ABB RobotStudio station: VInRoS_ROB_1_Project.rspag

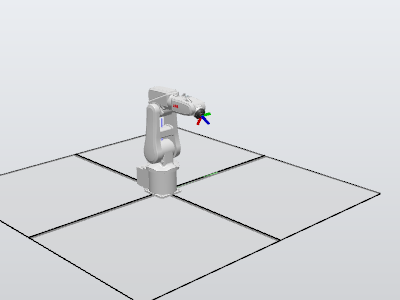
--- station ---
Station VInRoS_ROB_1_Project (saved by RobotStudio 23.2.10478.1)
Controller Controller1
  mechanical unit ROB_1: IRB120_3_58__01, 6 joints, base frame (0, 0, 0) mm
Layout (positions relative to the parent item):
  - IRB120_3_58__01 [mechanism, from %ABB.RobotStudio.Models.IRB120%\IRB120_3_58_G_01.rslib] at (0, 0, 0) mm; joint values [0, 0, 0, 0, 0.5236, 0] (rad or m)

--- Controller Data/Controller1/RAPID/TASK1/PROGMOD/Module1.mod ---
MODULE Module1
    ! ## =========================================================================== ##
    ! MIT License
    ! Copyright (c) 2021 Roman Parak
    ! Permission is hereby granted, free of charge, to any person obtaining a copy
    ! of this software and associated documentation files (the "Software"), to deal
    ! in the Software without restriction, including without limitation the rights
    ! to use, copy, modify, merge, publish, distribute, sublicense, and/or sell
    ! copies of the Software, and to permit persons to whom the Software is
    ! furnished to do so, subject to the following conditions:
    ! The above copyright notice and this permission notice shall be included in all
    ! copies or substantial portions of the Software.
    ! THE SOFTWARE IS PROVIDED "AS IS", WITHOUT WARRANTY OF ANY KIND, EXPRESS OR
    ! IMPLIED, INCLUDING BUT NOT LIMITED TO THE WARRANTIES OF MERCHANTABILITY,
    ! FITNESS FOR A PARTICULAR PURPOSE AND NONINFRINGEMENT. IN NO EVENT SHALL THE
    ! AUTHORS OR COPYRIGHT HOLDERS BE LIABLE FOR ANY CLAIM, DAMAGES OR OTHER
    ! LIABILITY, WHETHER IN AN ACTION OF CONTRACT, TORT OR OTHERWISE, ARISING FROM,
    ! OUT OF OR IN CONNECTION WITH THE SOFTWARE OR THE USE OR OTHER DEALINGS IN THE
    ! SOFTWARE.
    ! ## =========================================================================== ##
    ! Author   : Roman Parak
    ! Email    : Roman.Parak@outlook.com
    ! Github   : https://github.com/rparak
    ! File Name: T_ROB_MAIN_CTRL/Module1.mod
    ! ## =========================================================================== ##

    ! Description: !
    !   The main command structure for robot control !
    RECORD robot_command_main_str
        num start;
        num stop;
        num id;
        num update;
    ENDRECORD

    ! Description: !
    !   The main structure of the robot control parameters !
    RECORD robot_param_main_str
        num Trajectory_Size;
    ENDRECORD

    ! Description: !
    !   The main structure of robot status information !
    RECORD robot_status_str
        num in_position; ! Signaling when the robot is in the target position
        num active;      ! Signaling when everything on the robot's side is fine
        num id;          ! Identification number of the current state of the robot
        num update_done; ! Signaling when the parameter update is completed successfully
        num actual_trajectory_id;
    ENDRECORD

    ! Description: !
    !   The main structure of PLC status information !
    RECORD plc_status_str
        num active; ! Signaling when everything on the PC's (PLC) side is OK
        num update_done;
    ENDRECORD

    ! Description: !
    !   The main structure of status information !
    RECORD status_main_str
        plc_status_str plc;
        robot_status_str robot;
    ENDRECORD

    ! Description: !
    !   The main structure of internal values !
    RECORD internal_main_str
        num actual_state;               ! Current state in the main state machine
        num previous_state;             ! Previous state in the main state machine
        num accuracy_factor;            ! Accuracy factor for value conversion (Default)
        num accuracy_factor_QUATERNION; ! Accuracy factor for value conversion (QUATERNION)
        num actual_trajectory_id;
    ENDRECORD

    ! Description: !
    !   The main control structure of the robot !
    RECORD robot_ctrl_str
        robot_param_main_str parameter; ! Robot control parameters
        robot_command_main_str command; ! Command structure for robot control
        status_main_str status;         ! Robot status information
        internal_main_str internal;     ! Internal values
    ENDRECORD

    ! Call Main Structure
    PERS robot_ctrl_str rm_str;

    ! Joint Position Data
    PERS jointtarget J_Position{100};

    ! TCP Position Data
    PERS robtarget TCP_Position{100};

    ! Joint Speed Data
    PERS speeddata Speed{100};

    ! Joint Zone Data
    PERS zonedata Zone{100};

    ! Characteristics of a robotic tool (end-effector / gripper)
    PERS tooldata robTool;

    VAR num aux_trajectory_index_var;

    ! Description:               !
    !   Program Main Cycle:      !
    !       Type        : Normal !
    !       TrustLeve   : N/A    !
    !       Motion Task : YES    !
    PROC Main()
        TEST ROB_ST_MAIN_ID_PROFINET_OUT
            CASE 10: ! INITIALIZATION STATE !
                ! Description: !
                !   Initialization state to check everything on the PC's (PLC) side and activation to control !

                ! Initialize the internal value of the accuracy conversion factor
                rm_str.internal.accuracy_factor            := 100;
                rm_str.internal.accuracy_factor_QUATERNION := 100000000;

                SetDO ROB_ST_ACTIVE_PROFINET_OUT, 1;

                IF PLC_ST_ACTIVE_PROFINET_IN = 1 THEN
                    ! Wait State {rm_str.status.plc.ModuleOK = TRUE -> Everything on the PC's (PLC) side is OK}
                    SetGO ROB_ST_MAIN_ID_PROFINET_OUT, 20;
                ENDIF

            CASE 20: ! WAIT STATE !
                ! Description: !
                !   State of waiting for command with index from the PC's (PLC) !

                aux_trajectory_index_var := 0;

                IF PLC_CMD_START_PROFINET_IN = 1 AND PLC_CMD_MAIN_ID_PROFINET_IN = 1 THEN
                    SetDO ROB_ST_IN_POS_PROFINET_OUT, 0;
                    ! Move Joint (Absolute)
                    SetGO ROB_ST_MAIN_ID_PROFINET_OUT, 30;
                ELSEIF PLC_CMD_START_PROFINET_IN = 1 AND PLC_CMD_MAIN_ID_PROFINET_IN = 2 THEN
                    SetDO ROB_ST_IN_POS_PROFINET_OUT, 0;
                    ! Move Linear
                    SetGO ROB_ST_MAIN_ID_PROFINET_OUT, 40;
                ENDIF

                IF PLC_ST_ACTIVE_PROFINET_IN = 0 THEN
                    ! Initialization State {rm_str.PLC_ModuleOK = FALSE -> There is some problem with the PC's (PLC)}
                    SetGO ROB_ST_MAIN_ID_PROFINET_OUT, 10;
                ENDIF

            CASE 30: ! MOVE JOINT ABSOLUTE STATE - EXECUTE !
                ! Description: !
                !   Control Function (MoveAbsJ): Moves the robot to an absolute joint position !

                IF aux_trajectory_index_var = PLC_TRAJ_SIZE_PROFINET_IN THEN
                    SetDO ROB_ST_IN_POS_PROFINET_OUT, 1;
                    SetGO ROB_ST_MAIN_ID_PROFINET_OUT, 20;
                ELSE
                    SetGO ROB_MOTION_TRAJ_ID_PROFINET_OUT, aux_trajectory_index_var;
                    MoveAbsJ J_Position{aux_trajectory_index_var + 1}\NoEOffs, Speed{aux_trajectory_index_var + 1}, Zone{aux_trajectory_index_var + 1}, robTool\WObj:=wobj0;
                    aux_trajectory_index_var := aux_trajectory_index_var + 1;
                ENDIF

            CASE 40: ! MOVE CARTESIAN STATE - EXECUTE !
                ! Description: !
                !   Control Function (MoveL): Moves the tool center point (TCP) linearly !

                IF aux_trajectory_index_var = PLC_TRAJ_SIZE_PROFINET_IN THEN
                    SetDO ROB_ST_IN_POS_PROFINET_OUT, 1;
                    SetGO ROB_ST_MAIN_ID_PROFINET_OUT, 20;
                ELSE
                    SetGO ROB_MOTION_TRAJ_ID_PROFINET_OUT, aux_trajectory_index_var;
                    MoveL TCP_Position{aux_trajectory_index_var + 1}, Speed{aux_trajectory_index_var + 1}, Zone{aux_trajectory_index_var + 1}, robTool\WObj:=wobj0;
                    aux_trajectory_index_var := aux_trajectory_index_var + 1;
                ENDIF
        ENDTEST
    ENDPROC

    PROC ER_Reset_Parameters_MAIN_CTRL()
        ! Description:                                                   !
        !   Event routine function (non-parametric) for parameter reset. !
        !       Note: Configuration / Controller / Event Routine         !

        SetGO ROB_ST_MAIN_ID_PROFINET_OUT, 10;
        SetGO ROB_ST_UPT_ID_PROFINET_OUT, 10;

        ! Main Control Structure
        rm_str := [[0],[0,0,0,0],[[0,0],[0,0,0,0,0]],[0,0,0,0,0]];

        ! Characteristics of a robotic tool (end-effector / gripper)
        robTool := [TRUE,[[0,0,0],[1,0,0,0]],[0.001,[0,0,0.001],[1,0,0,0],0,0,0]];
	ENDPROC

    PROC ER_Reset_Parameters_Stopped()
        ! Description:                                                   !
        !   Event routine function (non-parametric) to reset parameters  !
        !   when the program is stopped.                                 !
        !       Note: Configuration / Controller / Event Routine         !

        SetDO ROB_ST_IN_POS_PROFINET_OUT, 1;
        SetGO ROB_ST_MAIN_ID_PROFINET_OUT, 10;
    ENDPROC
ENDMODULE

--- Controller Data/Controller1/RAPID/TASK2/PROGMOD/Module1.mod ---
MODULE Module1
    ! ## =========================================================================== ##
    ! MIT License
    ! Copyright (c) 2021 Roman Parak
    ! Permission is hereby granted, free of charge, to any person obtaining a copy
    ! of this software and associated documentation files (the "Software"), to deal
    ! in the Software without restriction, including without limitation the rights
    ! to use, copy, modify, merge, publish, distribute, sublicense, and/or sell
    ! copies of the Software, and to permit persons to whom the Software is
    ! furnished to do so, subject to the following conditions:
    ! The above copyright notice and this permission notice shall be included in all
    ! copies or substantial portions of the Software.
    ! THE SOFTWARE IS PROVIDED "AS IS", WITHOUT WARRANTY OF ANY KIND, EXPRESS OR
    ! IMPLIED, INCLUDING BUT NOT LIMITED TO THE WARRANTIES OF MERCHANTABILITY,
    ! FITNESS FOR A PARTICULAR PURPOSE AND NONINFRINGEMENT. IN NO EVENT SHALL THE
    ! AUTHORS OR COPYRIGHT HOLDERS BE LIABLE FOR ANY CLAIM, DAMAGES OR OTHER
    ! LIABILITY, WHETHER IN AN ACTION OF CONTRACT, TORT OR OTHERWISE, ARISING FROM,
    ! OUT OF OR IN CONNECTION WITH THE SOFTWARE OR THE USE OR OTHER DEALINGS IN THE
    ! SOFTWARE.
    ! ## =========================================================================== ##
    ! Author   : Roman Parak
    ! Email    : Roman.Parak@outlook.com
    ! Github   : https://github.com/rparak
    ! File Name: T_PLC_ROB_PROFINET/Module1.mod
    ! ## =========================================================================== ##


    ! Description: !
    !   The main command structure for robot control !
    RECORD robot_command_main_str
        num start;
        num stop;
        num id;
        num update;
    ENDRECORD

    ! Description: !
    !   The main structure of the robot control parameters !
    RECORD robot_param_main_str
        num Trajectory_Size;
    ENDRECORD

    ! Description: !
    !   The main structure of robot status information !
    RECORD robot_status_str
        num in_position; ! Signaling when the robot is in the target position
        num active;      ! Signaling when everything on the robot's side is fine
        num id;          ! Identification number of the current state of the robot
        num update_done; ! Signaling when the parameter update is completed successfully
        num actual_trajectory_id;
    ENDRECORD

    ! Description: !
    !   The main structure of PLC status information !
    RECORD plc_status_str
        num active; ! Signaling when everything on the PC's (PLC) side is OK
        num update_done;
    ENDRECORD

    ! Description: !
    !   The main structure of status information !
    RECORD status_main_str
        plc_status_str plc;
        robot_status_str robot;
    ENDRECORD

    ! Description: !
    !   The main structure of internal values !
    RECORD internal_main_str
        num actual_state;               ! Current state in the main state machine
        num previous_state;             ! Previous state in the main state machine
        num accuracy_factor;            ! Accuracy factor for value conversion (Default)
        num accuracy_factor_QUATERNION; ! Accuracy factor for value conversion (QUATERNION)
        num actual_trajectory_id;
    ENDRECORD

    ! Description: !
    !   The main control structure of the robot !
    RECORD robot_ctrl_str
        robot_param_main_str parameter; ! Robot control parameters
        robot_command_main_str command; ! Command structure for robot control
        status_main_str status;         ! Robot status information
        internal_main_str internal;     ! Internal values
    ENDRECORD

    ! Call Main Structure
    PERS robot_ctrl_str rm_str;

    ! Joint Position Data
    PERS jointtarget J_Position{100};

    ! TCP Position Data
    PERS robtarget TCP_Position{100};

    ! Joint Speed Data
    PERS speeddata Speed{100};

    ! Joint Zone Data
    PERS zonedata Zone{100};

    ! Characteristics of a robotic tool (end-effector / gripper)
    PERS tooldata robTool;

    ! Characteristics of a robotic tool (end-effector / gripper)
    !   Note: Current Data (T_ROB_PLC_PROFINET_CPR)
    PERS tooldata robTool_CPR;

    VAR num actual_traj_id;
    VAR num aux_traj_id;

    ! Mathematical Constant PI
    VAR num M_PI := 3.14159265358979323846264338327950288;

    VAR num update_state;

    ! Description:                   !
    !   Program Main Cycle:          !
    !       Type        : Semistatic !
    !       TrustLeve   : No Safety  !
    !       Motion Task : N/A        !
    PROC Main()
        TEST ROB_ST_UPT_ID_PROFINET_OUT
            CASE 10:
                actual_traj_id := 0;
                aux_traj_id    := 0;

                IF PLC_CMD_UTP_PROFINET_IN = 1 AND PLC_CMD_UPT_ID_PROFINET_IN = 1 THEN
                    ! Update Trajectory Parameters (Joint)
                    SetGO ROB_ST_UPT_ID_PROFINET_OUT, 40;
                ELSEIF PLC_CMD_UTP_PROFINET_IN = 1 AND PLC_CMD_UPT_ID_PROFINET_IN = 2 THEN
                    ! Update Trajectory Parameters (TCP)
                    SetGO ROB_ST_UPT_ID_PROFINET_OUT, 50;
                ELSEIF PLC_CMD_UTP_PROFINET_IN = 1 AND PLC_CMD_UPT_ID_PROFINET_IN = 10 THEN
                    ! Update Tool Parameters
                    SetGO ROB_ST_UPT_ID_PROFINET_OUT, 100;
                ENDIF

            CASE 40:
                IF PLC_TRAJ_SIZE_PROFINET_IN = actual_traj_id THEN
                    SetGO ROB_ST_UPT_ID_PROFINET_OUT, 10;
                ELSE
                    aux_traj_id := actual_traj_id;
                    SetGO ROB_ST_UPT_ID_PROFINET_OUT, 41;
                ENDIF

            CASE 41:
                IF actual_traj_id = aux_traj_id THEN
                    actual_traj_id := aux_traj_id + 1;
                    SetGO ROB_ST_UPT_ID_PROFINET_OUT, 42;
                ENDIF

            CASE 42:
                IF PLC_ST_UPDATE_DONE_PROFINET_IN = 1 THEN
                    SetDO ROB_ST_UPDATE_DONE_PROFINET_OUT, 0;
                    SetGO ROB_ST_UPT_ID_PROFINET_OUT, 43;
                ENDIF

            CASE 43:
                ! Set parameters for the specified motion type !
                ! SPEED / ZONE
                Speed{actual_traj_id} := set_speeddata(SPEED_DATA_PROFINET_IN); Zone{actual_traj_id} := set_zonedata(ZONE_DATA_PROFINET_IN);
                ! JOINT POSITION
                ! Q0 ... Q5
                J_Position{actual_traj_id}.robax.rax_1 := sign(Q0_SIGN_PROFINET_IN) * ((DnumToNum(GInputDnum(Q0_PROFINET_IN))) / rm_str.internal.accuracy_factor);
                J_Position{actual_traj_id}.robax.rax_2 := sign(Q1_SIGN_PROFINET_IN) * ((DnumToNum(GInputDnum(Q1_PROFINET_IN))) / rm_str.internal.accuracy_factor);
                J_Position{actual_traj_id}.robax.rax_3 := sign(Q2_SIGN_PROFINET_IN) * ((DnumToNum(GInputDnum(Q2_PROFINET_IN))) / rm_str.internal.accuracy_factor);
                J_Position{actual_traj_id}.robax.rax_4 := sign(Q3_SIGN_PROFINET_IN) * ((DnumToNum(GInputDnum(Q3_PROFINET_IN))) / rm_str.internal.accuracy_factor);
                J_Position{actual_traj_id}.robax.rax_5 := sign(Q4_SIGN_PROFINET_IN) * ((DnumToNum(GInputDnum(Q4_PROFINET_IN))) / rm_str.internal.accuracy_factor);
                J_Position{actual_traj_id}.robax.rax_6 := sign(Q5_SIGN_PROFINET_IN) * ((DnumToNum(GInputDnum(Q5_PROFINET_IN))) / rm_str.internal.accuracy_factor);
                ! Q0 - External
                J_Position{actual_traj_id}.extax.eax_a := sign(Q6_SIGN_PROFINET_IN) * ((DnumToNum(GInputDnum(Q6_PROFINET_IN))) / rm_str.internal.accuracy_factor);

                IF PLC_ST_UPDATE_DONE_PROFINET_IN = 0 THEN
                    SetDO ROB_ST_UPDATE_DONE_PROFINET_OUT, 1;
                    SetGO ROB_ST_UPT_ID_PROFINET_OUT, 40;
                ENDIF

            CASE 50:
                IF PLC_TRAJ_SIZE_PROFINET_IN = actual_traj_id THEN
                    SetGO ROB_ST_UPT_ID_PROFINET_OUT, 10;
                ELSE
                    aux_traj_id := actual_traj_id;
                    SetGO ROB_ST_UPT_ID_PROFINET_OUT, 51;
                ENDIF

            CASE 51:
                IF actual_traj_id = aux_traj_id THEN
                    actual_traj_id := aux_traj_id + 1;
                    SetGO ROB_ST_UPT_ID_PROFINET_OUT, 52;
                ENDIF

            CASE 52:
                IF PLC_ST_UPDATE_DONE_PROFINET_IN = 1 THEN
                    SetDO ROB_ST_UPDATE_DONE_PROFINET_OUT, 0;
                    SetGO ROB_ST_UPT_ID_PROFINET_OUT, 53;
                ENDIF

            CASE 53:
                ! Set parameters for the specified motion type !
                ! SPEED / ZONE
                Speed{actual_traj_id} := set_speeddata(SPEED_DATA_PROFINET_IN); Zone{actual_traj_id} := set_zonedata(ZONE_DATA_PROFINET_IN);
                ! TCP (Tool Center Point)
                ! Position
                TCP_Position{actual_traj_id}.trans.x := sign(TCP_POS_X_SIGN_PROFINET_IN) * ((DnumToNum(GInputDnum(TCP_POS_X_PROFINET_IN))) / rm_str.internal.accuracy_factor);
                TCP_Position{actual_traj_id}.trans.y := sign(TCP_POS_Y_SIGN_PROFINET_IN) * ((DnumToNum(GInputDnum(TCP_POS_Y_PROFINET_IN))) / rm_str.internal.accuracy_factor);
                TCP_Position{actual_traj_id}.trans.z := sign(TCP_POS_Z_SIGN_PROFINET_IN) * ((DnumToNum(GInputDnum(TCP_POS_Z_PROFINET_IN))) / rm_str.internal.accuracy_factor);
                ! Rotation
                TCP_Position{actual_traj_id}.rot := OrientZYX(sign(TCP_ROT_X_SIGN_PROFINET_IN) * ((DnumToNum(GInputDnum(TCP_ROT_X_PROFINET_IN))) / rm_str.internal.accuracy_factor),
                                                              sign(TCP_ROT_Y_SIGN_PROFINET_IN) * ((DnumToNum(GInputDnum(TCP_ROT_Y_PROFINET_IN))) / rm_str.internal.accuracy_factor),
                                                              sign(TCP_ROT_Z_SIGN_PROFINET_IN) * ((DnumToNum(GInputDnum(TCP_ROT_Z_PROFINET_IN))) / rm_str.internal.accuracy_factor));
                ! Configuration
                TCP_Position{actual_traj_id}.robconf.cf1 := sign(TCP_CFG_1_SIGN_PROFINET_IN) * (TCP_CFG_1_PROFINET_IN);
                TCP_Position{actual_traj_id}.robconf.cf4 := sign(TCP_CFG_4_SIGN_PROFINET_IN) * (TCP_CFG_4_PROFINET_IN);
                TCP_Position{actual_traj_id}.robconf.cf6 := sign(TCP_CFG_6_SIGN_PROFINET_IN) * (TCP_CFG_6_PROFINET_IN);
                TCP_Position{actual_traj_id}.robconf.cfx := sign(TCP_CFG_X_SIGN_PROFINET_IN) * (TCP_CFG_X_PROFINET_IN);
                ! External Position
                TCP_Position{actual_traj_id}.extax.eax_a := sign(TCP_EX_POS_SIGN_PROFINET_IN) * ((DnumToNum(GInputDnum(TCP_EX_POS_PROFINET_IN))) / rm_str.internal.accuracy_factor);

                IF PLC_ST_UPDATE_DONE_PROFINET_IN = 0 THEN
                    SetDO ROB_ST_UPDATE_DONE_PROFINET_OUT, 1;
                    SetGO ROB_ST_UPT_ID_PROFINET_OUT, 50;
                ENDIF

            CASE 100:! UPDATE TOOL PARAMETERS STATE !
                ! Description: !
                !   Define the parameters of the robotic tool                                            !

                ! The robot is holding the tool (TRUE / FALSE)
                IF RTOOL_RH_PROFINET_IN = 1 THEN
                    robTool.robhold := TRUE;
                ELSE
                    robTool.robhold := FALSE;
                ENDIF

                ! Translation position
                robTool.tframe.trans := [sign(RTOOL_X_POS_SING_PROFINET_IN) * ((DnumToNum(GInputDnum(RTOOL_X_POS_PROFINET_IN))) / rm_str.internal.accuracy_factor),
                                         sign(RTOOL_Y_POS_SING_PROFINET_IN) * ((DnumToNum(GInputDnum(RTOOL_Y_POS_PROFINET_IN))) / rm_str.internal.accuracy_factor),
                                         sign(RTOOL_Z_POS_SING_PROFINET_IN) * ((DnumToNum(GInputDnum(RTOOL_Z_POS_PROFINET_IN))) / rm_str.internal.accuracy_factor)];
                ! Rotation Position
                robTool.tframe.rot := [sign(RTOOL_QX_ROT_SIGN_PROFINET_IN) * ((DnumToNum(GInputDnum(RTOOL_QX_ROT_PROFINET_IN))) / rm_str.internal.accuracy_factor_QUATERNION),
                                       sign(RTOOL_QY_ROT_SIGN_PROFINET_IN) * ((DnumToNum(GInputDnum(RTOOL_QY_ROT_PROFINET_IN))) / rm_str.internal.accuracy_factor_QUATERNION),
                                       sign(RTOOL_QZ_ROT_SIGN_PROFINET_IN) * ((DnumToNum(GInputDnum(RTOOL_QZ_ROT_PROFINET_IN))) / rm_str.internal.accuracy_factor_QUATERNION),
                                       sign(RTOOL_QW_ROT_SIGN_PROFINET_IN) * ((DnumToNum(GInputDnum(RTOOL_QW_ROT_PROFINET_IN))) / rm_str.internal.accuracy_factor_QUATERNION)];
                ! Tool Mass
                robTool.tload.mass := GInput(RTOOL_MASS_PROFINET_IN) / rm_str.internal.accuracy_factor;

                ! Center of Gravity
                robTool.tload.cog := [sign(RTOOL_X_COG_SIGN_PROFINET_IN) * ((DnumToNum(GInputDnum(RTOOL_X_COG_PROFINET_IN))) / rm_str.internal.accuracy_factor),
                                      sign(RTOOL_Y_COG_SIGN_PROFINET_IN) * ((DnumToNum(GInputDnum(RTOOL_Y_COG_PROFINET_IN))) / rm_str.internal.accuracy_factor),
                                      sign(RTOOL_Z_COG_SIGN_PROFINET_IN) * ((DnumToNum(GInputDnum(RTOOL_Z_COG_PROFINET_IN))) / rm_str.internal.accuracy_factor)];
                ! Inertial axes of tool load
                robTool.tload.aom := [sign(RTOOL_QX_AOM_SIGN_PROFINET_IN) * ((DnumToNum(GInputDnum(RTOOL_QX_AOM_PROFINET_IN))) / rm_str.internal.accuracy_factor_QUATERNION),
                                      sign(RTOOL_QY_AOM_SIGN_PROFINET_IN) * ((DnumToNum(GInputDnum(RTOOL_QY_AOM_PROFINET_IN))) / rm_str.internal.accuracy_factor_QUATERNION),
                                      sign(RTOOL_QZ_AOM_SIGN_PROFINET_IN) * ((DnumToNum(GInputDnum(RTOOL_QZ_AOM_PROFINET_IN))) / rm_str.internal.accuracy_factor_QUATERNION),
                                      sign(RTOOL_QW_AOM_SIGN_PROFINET_IN) * ((DnumToNum(GInputDnum(RTOOL_QW_AOM_PROFINET_IN))) / rm_str.internal.accuracy_factor_QUATERNION)];
                ! Momets of inertia
                robTool.tload.ix := DnumToNum(GInputDnum(RTOOL_IX_MOI_PROFINET_IN)) / rm_str.internal.accuracy_factor;
                robTool.tload.iy := DnumToNum(GInputDnum(RTOOL_IY_MOI_PROFINET_IN)) / rm_str.internal.accuracy_factor;
                robTool.tload.iz := DnumToNum(GInputDnum(RTOOL_IZ_MOI_PROFINET_IN)) / rm_str.internal.accuracy_factor;

                ! Characteristics of a robotic tool (end-effector / gripper)
                !   Note: Upload (Current Data)
                robTool_CPR := robTool;

                ! The parameter update is completed successfully
                PulseDO ROB_ST_UPDATE_DONE_PROFINET_OUT;

                SetGO ROB_ST_UPT_ID_PROFINET_OUT, 10;
        ENDTEST
    ENDPROC

    FUNC num sign(num value)
        ! Description:                                                                !
        !   A simple mathematical function that extracts a sign from a digital value. !
        !                                                                             !
        ! IN:                                                                         !
        ! [1] value [num]: Digital Input (1 / 0).                                     !
        ! OUT:                                                                        !
        ! [1] return [num]: Sign (1: Positive {+}, -1: Negative {-}).                 !

        IF value = 1 THEN
           RETURN 1;
        ELSE
           RETURN -1;
        ENDIF
    ENDFUNC

    FUNC num RadToDeg(num value)
        ! Description:                                       !
        !   Conversion function between radians and degrees. !
        !                                                    !
        ! IN:                                                !
        ! [1] value [num]: Real number (Radian).             !
        ! OUT:                                               !
        ! [1] return [num]: Degree.                          !

        RETURN ((value) * 180.0 / M_PI);
    ENDFUNC

    FUNC speeddata set_speeddata(num value)
        ! Description:                                                                                               !
        !   The function to specify the velocity at which both the robot and the external axes move.                 !
        !                                                                                                            !
        ! IN:                                                                                                        !
        ! [1] value [num]: Specified value from the PC's (PLC).                                                      !
        ! OUT:                                                                                                       !
        ! [1] return [speeddata {Velocity: TCP, Orientation, Linear External Axes, Rotational External Axes}]:
        !                              Predefined speed data to be used for moving the robot and the external axes . !

        TEST value
            CASE 0:
                RETURN [5, 50, 1000, 500];
            CASE 1:
                RETURN [10, 50, 1000, 500];
            CASE 2:
                RETURN [20, 50, 1000, 500];
            CASE 3:
                RETURN [30, 50, 1000, 500];
            CASE 4:
                RETURN [40, 100, 1000, 500];
            CASE 5:
                RETURN [50, 100, 1000, 500];
            CASE 6:
                RETURN [60, 100, 1000, 500];
            CASE 7:
                RETURN [80, 100, 1000, 500];
            CASE 8:
                RETURN [100, 200, 1000, 500];
            CASE 9:
                RETURN [150, 200, 1000, 500];
            CASE 10:
                RETURN [200, 200, 1000, 500];
            CASE 11:
                RETURN [300, 200, 1000, 500];
            CASE 12:
                RETURN [400, 300, 1000, 500];
            CASE 13:
                RETURN [500, 300, 1000, 500];
            CASE 14:
                RETURN [600, 300, 1000, 500];
            CASE 15:
                RETURN [800, 300, 1000, 500];
            CASE 16:
                RETURN [1000, 400, 1000, 500];
            CASE 17:
                RETURN [1500, 400, 1000, 500];
            CASE 18:
                RETURN [2000, 400, 1000, 500];
            CASE 19:
                RETURN [2500, 400, 1000, 500];
            CASE 20:
                RETURN [3000, 500, 1000, 500];
            CASE 21:
                RETURN [4000, 500, 1000, 500];
            CASE 22:
                RETURN [5000, 500, 1000, 500];
            CASE 23:
                RETURN [6000, 500, 1000, 500];
        ENDTEST
    ENDFUNC

    FUNC zonedata set_zonedata(num value)
        ! Description:                                                                                            !
        !   The function to specify how a position is to be terminated, i.e. how close to the programmed position
        !   the axes must be before moving towards the next position.                                             !
        !                                                                                                         !
        ! IN:                                                                                                     !
        ! [1] value [num]: Specified value from the PC's (PLC).                                                   !
        ! OUT:                                                                                                    !
        ! [1] return [zonedata]: Defines whether the movement is to terminate as a stop point (fine point) or
        !                        as a fly-by point.                                                               !
        !                           Stop points : Use zonedata named fine.                                        !
        !                           Other       : Fly-by points(z0 {0.3 mm / 0.03?} .. z200 {200 mm / 30?})       !

        TEST value
            CASE 0:
                RETURN fine;
            CASE 1:
                RETURN z0;
            CASE 2:
                RETURN z1;
            CASE 3:
                RETURN z5;
            CASE 4:
                RETURN z10;
            CASE 5:
                RETURN z15;
            CASE 6:
                RETURN z20;
            CASE 7:
                RETURN z30;
            CASE 8:
                RETURN z40;
            CASE 9:
                RETURN z50;
            CASE 10:
                RETURN z60;
            CASE 11:
                RETURN z80;
            CASE 12:
                RETURN z100;
            CASE 13:
                RETURN z150;
            CASE 14:
                RETURN z200;
        ENDTEST
    ENDFUNC
ENDMODULE

--- Controller Data/Controller1/RAPID/TASK3/PROGMOD/Module1.mod ---
MODULE Module1
    ! ## =========================================================================== ##
    ! MIT License
    ! Copyright (c) 2021 Roman Parak
    ! Permission is hereby granted, free of charge, to any person obtaining a copy
    ! of this software and associated documentation files (the "Software"), to deal
    ! in the Software without restriction, including without limitation the rights
    ! to use, copy, modify, merge, publish, distribute, sublicense, and/or sell
    ! copies of the Software, and to permit persons to whom the Software is
    ! furnished to do so, subject to the following conditions:
    ! The above copyright notice and this permission notice shall be included in all
    ! copies or substantial portions of the Software.
    ! THE SOFTWARE IS PROVIDED "AS IS", WITHOUT WARRANTY OF ANY KIND, EXPRESS OR
    ! IMPLIED, INCLUDING BUT NOT LIMITED TO THE WARRANTIES OF MERCHANTABILITY,
    ! FITNESS FOR A PARTICULAR PURPOSE AND NONINFRINGEMENT. IN NO EVENT SHALL THE
    ! AUTHORS OR COPYRIGHT HOLDERS BE LIABLE FOR ANY CLAIM, DAMAGES OR OTHER
    ! LIABILITY, WHETHER IN AN ACTION OF CONTRACT, TORT OR OTHERWISE, ARISING FROM,
    ! OUT OF OR IN CONNECTION WITH THE SOFTWARE OR THE USE OR OTHER DEALINGS IN THE
    ! SOFTWARE.
    ! ## =========================================================================== ##
    ! Author   : Roman Parak
    ! Email    : Roman.Parak@outlook.com
    ! Github   : https://github.com/rparak
    ! File Name: T_ROB_PLC_PROFINET_Q/Module1.mod
    ! ## =========================================================================== ##


    ! Description: !
    !   Joint Position Data (Q0 - Q5): sign (+-) !
    RECORD robot_data_joint_sign_str
        num Q0;
        num Q1;
        num Q2;
        num Q3;
        num Q4;
        num Q5;
        num Q6;
    ENDRECORD

    ! Description: !
    !   The main structure of data collection on the current position of the robot with sign (+-) !
    RECORD robot_data_main_str
        robot_data_joint_sign_str Joint_Sign; ! Joint Position Data (Q0 - Q6): sign (+-)
        jointtarget JOINT_CURRENT_DATA;       ! Joint Position Data
    ENDRECORD

    ! Call Main Structure
    !   Note: VAR robot_dataC_main_str r_data_collection := [[0,0,0,0,0,0,0],[[0,0,0,0,0,0],[0,0,0,0,0,0]]];
    VAR robot_data_main_str r_data;

    ! Characteristics of a robotic tool (end-effector / gripper)
    !   Note: Current Data (T_ROB_PLC_PROFINET_CPR)
    !PERS tooldata robTool_CPR := [TRUE,[[0,0,0],[1,0,0,0]],[0.001,[0,0,0.001],[1,0,0,0],0,0,0]];
    PERS tooldata robTool_CPR;

    ! Variable for rounded (Joint, Cartesian) data
    VAR num NUM_OF_ROUNDED_PLACES := 2;

    ! Mathematical Constant PI
    VAR num M_PI := 3.14159;

    ! Accuracy factor for value conversion
    VAR num accuracy_factor := 100;

    ! Description:                   !
    !   Program Main Cycle:          !
    !       Type        : Semistatic !
    !       TrustLeve   : No Safety  !
    !       Motion Task : N/A        !
    PROC Main()
        ! Description:                                                       !
        !   Read the current angles of the robot axes (Joint).               !
        !       Note: The resulting data is rounded with the Round function  !

        r_data.JOINT_CURRENT_DATA := CJointT();

        ! Joint (Q0 .. Q5) -> Q0 Parameter (Joint Number 0)
        r_data.Joint_Sign.Q0 := sign(Round(r_data.JOINT_CURRENT_DATA.robax.rax_1 \Dec:=NUM_OF_ROUNDED_PLACES));
        SetDo Q0_SIGN_PROFINET_OUT, r_data.Joint_Sign.Q0;
        IF r_data.Joint_Sign.Q0 = 0 THEN
            SetGO Q0_PROFINET_OUT, Round(((-1) * (r_data.JOINT_CURRENT_DATA.robax.rax_1 * accuracy_factor)) \Dec:=0);
        ELSE
            SetGO Q0_PROFINET_OUT, Round((r_data.JOINT_CURRENT_DATA.robax.rax_1 * accuracy_factor) \Dec:=0);
        ENDIF
        !   Q0 Parameter (External)
        r_data.Joint_Sign.Q6 := sign(Round(r_data.JOINT_CURRENT_DATA.extax.eax_a \Dec:=NUM_OF_ROUNDED_PLACES));
        SetDo Q6_SIGN_PROFINET_OUT, r_data.Joint_Sign.Q6;
        IF r_data.JOINT_CURRENT_DATA.extax.eax_a <> 9E+09 THEN
            IF r_data.Joint_Sign.Q6 = 0 THEN
                SetGO Q6_PROFINET_OUT, Round(((-1) * (r_data.JOINT_CURRENT_DATA.extax.eax_a * accuracy_factor)) \Dec:=0);
            ELSE
                SetGO Q6_PROFINET_OUT, Round((r_data.JOINT_CURRENT_DATA.extax.eax_a * accuracy_factor) \Dec:=0);
            ENDIF
        ENDIF

        ! Joint (Q0 .. Q5) -> Q1 Parameter (Joint Number 1)
        r_data.Joint_Sign.Q1 := sign(Round(r_data.JOINT_CURRENT_DATA.robax.rax_2 \Dec:=NUM_OF_ROUNDED_PLACES));
        SetDo Q1_SIGN_PROFINET_OUT, r_data.Joint_Sign.Q1;
        IF r_data.Joint_Sign.Q1 = 0 THEN
            SetGO Q1_PROFINET_OUT, Round(((-1) * (r_data.JOINT_CURRENT_DATA.robax.rax_2 * accuracy_factor)) \Dec:=0);
        ELSE
            SetGO Q1_PROFINET_OUT, Round((r_data.JOINT_CURRENT_DATA.robax.rax_2 * accuracy_factor) \Dec:=0);
        ENDIF

        ! Joint (Q0 .. Q5) -> Q2 Parameter (Joint Number 2)
        r_data.Joint_Sign.Q2 := sign(Round(r_data.JOINT_CURRENT_DATA.robax.rax_3 \Dec:=NUM_OF_ROUNDED_PLACES));
        SetDo Q2_SIGN_PROFINET_OUT, r_data.Joint_Sign.Q2;
        IF r_data.Joint_Sign.Q2 = 0 THEN
            SetGO Q2_PROFINET_OUT, Round(((-1) * (r_data.JOINT_CURRENT_DATA.robax.rax_3 * accuracy_factor)) \Dec:=0);
        ELSE
            SetGO Q2_PROFINET_OUT, Round((r_data.JOINT_CURRENT_DATA.robax.rax_3 * accuracy_factor) \Dec:=0);
        ENDIF

        ! Joint (Q0 .. Q5) -> Q3 Parameter (Joint Number 3)
        r_data.Joint_Sign.Q3 := sign(Round(r_data.JOINT_CURRENT_DATA.robax.rax_4 \Dec:=NUM_OF_ROUNDED_PLACES));
        SetDo Q3_SIGN_PROFINET_OUT, r_data.Joint_Sign.Q3;
        IF r_data.Joint_Sign.Q3 = 0 THEN
            SetGO Q3_PROFINET_OUT, Round(((-1) * (r_data.JOINT_CURRENT_DATA.robax.rax_4 * accuracy_factor)) \Dec:=0);
        ELSE
            SetGO Q3_PROFINET_OUT, Round((r_data.JOINT_CURRENT_DATA.robax.rax_4 * accuracy_factor) \Dec:=0);
        ENDIF

        ! Joint (Q0 .. Q5) -> Q4 Parameter (Joint Number 4)
        r_data.Joint_Sign.Q4 := sign(Round(r_data.JOINT_CURRENT_DATA.robax.rax_5 \Dec:=NUM_OF_ROUNDED_PLACES));
        SetDo Q4_SIGN_PROFINET_OUT, r_data.Joint_Sign.Q4;
        IF r_data.Joint_Sign.Q4 = 0 THEN
            SetGO Q4_PROFINET_OUT, Round(((-1) * (r_data.JOINT_CURRENT_DATA.robax.rax_5 * accuracy_factor)) \Dec:=0);
        ELSE
            SetGO Q4_PROFINET_OUT, Round((r_data.JOINT_CURRENT_DATA.robax.rax_5 * accuracy_factor) \Dec:=0);
        ENDIF

        ! Joint (Q0 .. Q5) -> Q5 Parameter (Joint Number 5)
        r_data.Joint_Sign.Q5 := sign(Round(r_data.JOINT_CURRENT_DATA.robax.rax_6 \Dec:=NUM_OF_ROUNDED_PLACES));
        SetDo Q5_SIGN_PROFINET_OUT, r_data.Joint_Sign.Q5;
        IF r_data.Joint_Sign.Q5 = 0 THEN
            SetGO Q5_PROFINET_OUT, Round(((-1) * (r_data.JOINT_CURRENT_DATA.robax.rax_6 * accuracy_factor)) \Dec:=0);
        ELSE
            SetGO Q5_PROFINET_OUT, Round((r_data.JOINT_CURRENT_DATA.robax.rax_6 * accuracy_factor) \Dec:=0);
        ENDIF
    ENDPROC

    FUNC num sign(num value)
        ! Description:                                                       !
        !   A simple mathematical function that extracts a real number sign. !
        !                                                                    !
        ! IN:                                                                !
        ! [1] value [num]: Real number.                                      !
        ! OUT:                                                               !
        ! [1] return [num]: Sign (1: Positive {+}, 0: Negative {-}).         !

        IF value >= 0 THEN
           RETURN 1;
        ELSE
           RETURN 0;
        ENDIF
    ENDFUNC

    PROC ER_Reset_Parameters_Q()
        ! Description:                                                   !
        !   Event routine function (non-parametric) for parameter reset. !
        !       Note: Configuration / Controller / Event Routine         !

        ! Main Structure for data collection
        r_data := [[0,0,0,0,0,0,0],[[0,0,0,0,0,0],[0,0,0,0,0,0]]];

        ! Characteristics of a robotic tool (end-effector / gripper)
        robTool_CPR := [TRUE,[[0,0,0],[1,0,0,0]],[0.001,[0,0,0.001],[1,0,0,0],0,0,0]];
	ENDPROC
ENDMODULE

--- Controller Data/Controller1/RAPID/TASK4/PROGMOD/Module1.mod ---
MODULE Module1
    ! Description: !
    !   TCP (Configuration - 1, 4, 6, X) !
    RECORD robot_data_tcp_cfg_sign_str
        num Cfg_1;
        num Cfg_4;
        num Cfg_6;
        num Cfg_X;
    ENDRECORD

    ! Description: !
    !   TCP (Position, Rotation - X, Y, Z) !
    RECORD robot_data_tcp_pr_sign_str
        num X;
        num Y;
        num Z;
    ENDRECORD

    ! Description: !
    !   TCP (Position, Rotation, Configuration): sign (+-) !
    RECORD robot_data_tcp_sign_str
        robot_data_tcp_pr_sign_str Position;
        robot_data_tcp_pr_sign_str Rotation;
        robot_data_tcp_cfg_sign_str Configuration;
        num External_Position;
    ENDRECORD

    ! Description: !
    !   The main structure of data collection on the current position of the robot with sign (+-) !
    RECORD robot_data_main_str
        robot_data_tcp_sign_str TCP_Sign; ! TCP (Position, Rotation - X, Y, Z): sign (+-)
        robtarget ROB_CURRENT_DATA;       ! Position Data (Cartesian)
    ENDRECORD

    ! Call Main Structure
    !   Note: VAR robot_dataC_main_str r_data := [[[0,0,0],[0,0,0],[0,0,0,0],0],[[0,0,0],[0,0,0,0],[0,0,0,0],[0,0,0,0,0,0]]];;
    VAR robot_data_main_str r_data;

    ! Characteristics of a robotic tool (end-effector / gripper)
    !   Note: Current Data (T_ROB_PLC_PROFINET_CPR)
    !PERS tooldata robTool_CPR := [TRUE,[[0,0,0],[1,0,0,0]],[0.001,[0,0,0.001],[1,0,0,0],0,0,0]];
    PERS tooldata robTool_CPR;

    ! Variable for rounded (Joint, Cartesian) data
    VAR num NUM_OF_ROUNDED_PLACES := 2;

    ! Mathematical Constant PI
    VAR num M_PI := 3.14159;

    ! Accuracy factor for value conversion
    VAR num accuracy_factor := 100;
    VAR robtarget a;

    ! Description:                   !
    !   Program Main Cycle:          !
    !       Type        : Semistatic !
    !       TrustLeve   : No Safety  !
    !       Motion Task : N/A        !
    PROC Main()
        ! Description:                                                       !
        !   Read the the current Tool Center Point (TCP) of the robot.       !
        !       Note: The resulting data is rounded with the Round function  !

        r_data.ROB_CURRENT_DATA := CRobT(\Tool:=robTool_CPR \WObj:=wobj0);

        ! TCP Position (X, Y, Z) -> X Parameter
        r_data.TCP_Sign.Position.X := sign(Round(r_data.ROB_CURRENT_DATA.trans.x \Dec:=NUM_OF_ROUNDED_PLACES));
        SetDO TCP_POS_X_SIGN_PROFINET_OUT, r_data.TCP_Sign.Position.X;
        IF r_data.TCP_Sign.Position.X = 0 THEN
            SetGO TCP_POS_X_PROFINET_OUT, Round(((-1) * (r_data.ROB_CURRENT_DATA.trans.x * accuracy_factor)) \Dec:=0);
        ELSE
            SetGO TCP_POS_X_PROFINET_OUT, Round((r_data.ROB_CURRENT_DATA.trans.x * accuracy_factor) \Dec:=0);
        ENDIF

        ! TCP Position (X, Y, Z) -> Y Parameter
        r_data.TCP_Sign.Position.Y := sign(Round(r_data.ROB_CURRENT_DATA.trans.y \Dec:=NUM_OF_ROUNDED_PLACES));
        SetDO TCP_POS_Y_SIGN_PROFINET_OUT, r_data.TCP_Sign.Position.Y;
        IF r_data.TCP_Sign.Position.Y = 0 THEN
            SetGO TCP_POS_Y_PROFINET_OUT, Round(((-1) * (r_data.ROB_CURRENT_DATA.trans.y * accuracy_factor)) \Dec:=0);
        ELSE
            SetGO TCP_POS_Y_PROFINET_OUT, Round((r_data.ROB_CURRENT_DATA.trans.y * accuracy_factor) \Dec:=0);
        ENDIF

        ! TCP Position (X, Y, Z) -> Z Parameter
        r_data.TCP_Sign.Position.Z := sign(Round(r_data.ROB_CURRENT_DATA.trans.z \Dec:=NUM_OF_ROUNDED_PLACES));
        SetDO TCP_POS_Z_SIGN_PROFINET_OUT, r_data.TCP_Sign.Position.Z;
        IF r_data.TCP_Sign.Position.Z = 0 THEN
            SetGO TCP_POS_Z_PROFINET_OUT, Round(((-1) * (r_data.ROB_CURRENT_DATA.trans.z * accuracy_factor)) \Dec:=0);
        ELSE
            SetGO TCP_POS_Z_PROFINET_OUT, Round((r_data.ROB_CURRENT_DATA.trans.z * accuracy_factor) \Dec:=0);
        ENDIF

        ! Description:                                                                    !
        !   Calculation of EA (Euler Angles) from quaternions using the EulerZYX function !

        ! TCP Rotation (Euler Angles: X, Y, Z) -> X Parameter
        r_data.TCP_Sign.Rotation.X := sign(Round(EulerZYX(\X, r_data.ROB_CURRENT_DATA.rot) \Dec:=NUM_OF_ROUNDED_PLACES));
        SetDO TCP_ROT_X_SIGN_PROFINET_OUT, r_data.TCP_Sign.Rotation.X;
        IF r_data.TCP_Sign.Rotation.X = 0 THEN
            SetGO TCP_ROT_X_PROFINET_OUT, Round(((-1) * (EulerZYX(\X, r_data.ROB_CURRENT_DATA.rot) * accuracy_factor)) \Dec:=0);
        ELSE
            SetGO TCP_ROT_X_PROFINET_OUT, Round((EulerZYX(\X, r_data.ROB_CURRENT_DATA.rot) * accuracy_factor) \Dec:=0);
        ENDIF

        ! TCP Rotation (Euler Angles: X, Y, Z) -> Y Parameter
        r_data.TCP_Sign.Rotation.Y := sign(Round(EulerZYX(\Y, r_data.ROB_CURRENT_DATA.rot) \Dec:=NUM_OF_ROUNDED_PLACES));
        SetDO TCP_ROT_Y_SIGN_PROFINET_OUT, r_data.TCP_Sign.Rotation.Y;
        IF r_data.TCP_Sign.Rotation.Y = 0 THEN
            SetGO TCP_ROT_Y_PROFINET_OUT, Round(((-1) * (EulerZYX(\Y, r_data.ROB_CURRENT_DATA.rot) * accuracy_factor)) \Dec:=0);
        ELSE
            SetGO TCP_ROT_Y_PROFINET_OUT, Round((EulerZYX(\Y, r_data.ROB_CURRENT_DATA.rot) * accuracy_factor) \Dec:=0);
        ENDIF

        ! TCP Rotation (Euler Angles: X, Y, Z) -> Z Parameter
        r_data.TCP_Sign.Rotation.Z := sign(Round(EulerZYX(\Z, r_data.ROB_CURRENT_DATA.rot) \Dec:=NUM_OF_ROUNDED_PLACES));
        SetDO TCP_ROT_Z_SIGN_PROFINET_OUT, r_data.TCP_Sign.Rotation.Z;
        IF r_data.TCP_Sign.Rotation.Z = 0 THEN
            SetGO TCP_ROT_Z_PROFINET_OUT, Round(((-1) * (EulerZYX(\Z, r_data.ROB_CURRENT_DATA.rot) * accuracy_factor)) \Dec:=0);
        ELSE
            SetGO TCP_ROT_Z_PROFINET_OUT, Round((EulerZYX(\Z, r_data.ROB_CURRENT_DATA.rot) * accuracy_factor) \Dec:=0);
        ENDIF

        ! Description:                                             !
        !   Expression of the configuration: Cfg -> 1, 4, 6, and X !

        ! TCP Configuration (1, 4, 6, X) -> Parameter 1
        r_data.TCP_Sign.Configuration.Cfg_1 := sign(r_data.ROB_CURRENT_DATA.robconf.cf1);
        SetDO TCP_CFG_1_SIGN_PROFINET_OUT, r_data.TCP_Sign.Configuration.Cfg_1;
        IF r_data.TCP_Sign.Configuration.Cfg_1 = 0 THEN
            SetGO TCP_CFG_1_PROFINET_OUT, (-1) * r_data.ROB_CURRENT_DATA.robconf.cf1;
        ELSE
            SetGO TCP_CFG_1_PROFINET_OUT, r_data.ROB_CURRENT_DATA.robconf.cf1;
        ENDIF

        ! TCP Configuration (1, 4, 6, X) -> Parameter 4
        r_data.TCP_Sign.Configuration.Cfg_4 := sign(r_data.ROB_CURRENT_DATA.robconf.cf4);
        SetDO TCP_CFG_4_SIGN_PROFINET_OUT, r_data.TCP_Sign.Configuration.Cfg_4;
        IF r_data.TCP_Sign.Configuration.Cfg_4 = 0 THEN
            SetGO TCP_CFG_4_PROFINET_OUT, (-1) * r_data.ROB_CURRENT_DATA.robconf.cf4;
        ELSE
            SetGO TCP_CFG_4_PROFINET_OUT, r_data.ROB_CURRENT_DATA.robconf.cf4;
        ENDIF

        ! TCP Configuration (1, 4, 6, X) -> Parameter 6
        r_data.TCP_Sign.Configuration.Cfg_6 := sign(r_data.ROB_CURRENT_DATA.robconf.cf6);
        SetDO TCP_CFG_6_SIGN_PROFINET_OUT, r_data.TCP_Sign.Configuration.Cfg_6;
        IF r_data.TCP_Sign.Configuration.Cfg_6 = 0 THEN
            SetGO TCP_CFG_6_PROFINET_OUT, (-1) * r_data.ROB_CURRENT_DATA.robconf.cf6;
        ELSE
            SetGO TCP_CFG_6_PROFINET_OUT, r_data.ROB_CURRENT_DATA.robconf.cf6;
        ENDIF

        ! TCP Configuration (1, 4, 6, X) -> Parameter X
        r_data.TCP_Sign.Configuration.Cfg_X := sign(r_data.ROB_CURRENT_DATA.robconf.cfx);
        SetDO TCP_CFG_X_SIGN_PROFINET_OUT, r_data.TCP_Sign.Configuration.Cfg_X;
        IF r_data.TCP_Sign.Configuration.Cfg_X = 0 THEN
            SetGO TCP_CFG_X_PROFINET_OUT, (-1) * r_data.ROB_CURRENT_DATA.robconf.cfx;
        ELSE
            SetGO TCP_CFG_X_PROFINET_OUT, r_data.ROB_CURRENT_DATA.robconf.cfx;
        ENDIF

        ! Description:                      !
        !   Expression of the external axis !

        ! TCP External Axis Position
        r_data.TCP_Sign.External_Position := sign(Round(r_data.ROB_CURRENT_DATA.extax.eax_a \Dec:=NUM_OF_ROUNDED_PLACES));
        SetDO TCP_EX_POS_SIGN_PROFINET_OUT, r_data.TCP_Sign.External_Position;
        IF r_data.ROB_CURRENT_DATA.extax.eax_a <> 9E+09 THEN
            IF r_data.TCP_Sign.External_Position = 0 THEN
                SetGO TCP_EX_POS_PROFINET_OUT, Round(((-1) * (r_data.ROB_CURRENT_DATA.extax.eax_a * accuracy_factor)) \Dec:=0);
            ELSE
                SetGO TCP_EX_POS_PROFINET_OUT, Round((r_data.ROB_CURRENT_DATA.extax.eax_a * accuracy_factor) \Dec:=0);
            ENDIF
        ENDIF

    ENDPROC

    FUNC num sign(num value)
        ! Description:                                                       !
        !   A simple mathematical function that extracts a real number sign. !
        !                                                                    !
        ! IN:                                                                !
        ! [1] value [num]: Real number.                                      !
        ! OUT:                                                               !
        ! [1] return [num]: Sign (1: Positive {+}, 0: Negative {-}).         !

        IF value >= 0 THEN
           RETURN 1;
        ELSE
           RETURN 0;
        ENDIF
    ENDFUNC

    PROC ER_Reset_Parameters_TCP()
        ! Description:                                                   !
        !   Event routine function (non-parametric) for parameter reset. !
        !       Note: Configuration / Controller / Event Routine         !

        ! Main Structure for data collection
        r_data := [[[0,0,0],[0,0,0],[0,0,0,0],0],[[0,0,0],[0,0,0,0],[0,0,0,0],[0,0,0,0,0,0]]];

        ! Characteristics of a robotic tool (end-effector / gripper)
        robTool_CPR := [TRUE,[[0,0,0],[1,0,0,0]],[0.001,[0,0,0.001],[1,0,0,0],0,0,0]];
	ENDPROC
ENDMODULE

--- Controller Data/Controller1/SYSPAR/EIO.cfg ---
EIO:CFG_1.0:6:1::
#
INDUSTRIAL_NETWORK:

      -Name "PROFINET" -Connection "PROFINET Network"\
      -Label "PROFINET Controller/Device Network" -StationName ""
#
PROFINET_DRIVER:

      -Name "PROFINET_COMMON_DATA"
#
PROFINET_INTERNAL_DEVICE:

      -Name "PN_Internal_Device" -VendorName "ABB Robotics"\
      -ProductName "PROFINET Internal Device" -OutputSize 256 -InputSize 256\
      -HostDevice "PN_Internal_Device"
#
EIO_SIGNAL:

      -Name "ROB_ST_ACTIVE_PROFINET_OUT" -SignalType "DO"\
      -Device "PN_Internal_Device" -DeviceMap "0" -EncType "UNSIGNED"

      -Name "ROB_ST_UPDATE_DONE_PROFINET_OUT" -SignalType "DO"\
      -Device "PN_Internal_Device" -DeviceMap "1" -EncType "UNSIGNED"

      -Name "ROB_ST_IN_POS_PROFINET_OUT" -SignalType "DO"\
      -Device "PN_Internal_Device" -DeviceMap "2" -EncType "UNSIGNED"

      -Name "SYS_MOTOR_ON_PROFINET_OUT" -SignalType "DO"\
      -Device "PN_Internal_Device" -DeviceMap "8" -EncType "UNSIGNED"

      -Name "SYS_MOTOR_OFF_PROFINET_OUT" -SignalType "DO"\
      -Device "PN_Internal_Device" -DeviceMap "9" -EncType "UNSIGNED"

      -Name "SYS_PP_MOVED_PROFINET_OUT" -SignalType "DO"\
      -Device "PN_Internal_Device" -DeviceMap "10" -EncType "UNSIGNED"

      -Name "SYS_CYCLE_ON_PROFINET_OUT" -SignalType "DO"\
      -Device "PN_Internal_Device" -DeviceMap "11" -EncType "UNSIGNED"

      -Name "ROB_ST_UPT_ID_PROFINET_OUT" -SignalType "GO"\
      -Device "PN_Internal_Device" -DeviceMap "16-23" -EncType "UNSIGNED"

      -Name "ROB_ST_MAIN_ID_PROFINET_OUT" -SignalType "GO"\
      -Device "PN_Internal_Device" -DeviceMap "24-31" -EncType "UNSIGNED"

      -Name "Q0_PROFINET_OUT" -SignalType "GO" -Device "PN_Internal_Device"\
      -DeviceMap "48-63" -EncType "UNSIGNED"

      -Name "Q1_PROFINET_OUT" -SignalType "GO" -Device "PN_Internal_Device"\
      -DeviceMap "64-79" -EncType "UNSIGNED"

      -Name "Q2_PROFINET_OUT" -SignalType "GO" -Device "PN_Internal_Device"\
      -DeviceMap "80-95" -EncType "UNSIGNED"

      -Name "Q3_PROFINET_OUT" -SignalType "GO" -Device "PN_Internal_Device"\
      -DeviceMap "96-111" -EncType "UNSIGNED"

      -Name "Q4_PROFINET_OUT" -SignalType "GO" -Device "PN_Internal_Device"\
      -DeviceMap "112-127" -EncType "UNSIGNED"

      -Name "Q5_PROFINET_OUT" -SignalType "GO" -Device "PN_Internal_Device"\
      -DeviceMap "128-143" -EncType "UNSIGNED"

      -Name "Q0_SIGN_PROFINET_OUT" -SignalType "DO" -Device "PN_Internal_Device"\
      -DeviceMap "160" -EncType "UNSIGNED"

      -Name "Q1_SIGN_PROFINET_OUT" -SignalType "DO" -Device "PN_Internal_Device"\
      -DeviceMap "161" -EncType "UNSIGNED"

      -Name "Q2_SIGN_PROFINET_OUT" -SignalType "DO" -Device "PN_Internal_Device"\
      -DeviceMap "162" -EncType "UNSIGNED"

      -Name "Q3_SIGN_PROFINET_OUT" -SignalType "DO" -Device "PN_Internal_Device"\
      -DeviceMap "163" -EncType "UNSIGNED"

      -Name "Q4_SIGN_PROFINET_OUT" -SignalType "DO" -Device "PN_Internal_Device"\
      -DeviceMap "164" -EncType "UNSIGNED"

      -Name "Q5_SIGN_PROFINET_OUT" -SignalType "DO" -Device "PN_Internal_Device"\
      -DeviceMap "165" -EncType "UNSIGNED"

      -Name "PLC_ST_ACTIVE_PROFINET_IN" -SignalType "DI"\
      -Device "PN_Internal_Device" -DeviceMap "0"

      -Name "PLC_ST_UPDATE_DONE_PROFINET_IN" -SignalType "DI"\
      -Device "PN_Internal_Device" -DeviceMap "1"

      -Name "SYS_MOTOR_ON_PROFINET_IN" -SignalType "DI"\
      -Device "PN_Internal_Device" -DeviceMap "8"

      -Name "SYS_MOTOR_OFF_PROFINET_IN" -SignalType "DI"\
      -Device "PN_Internal_Device" -DeviceMap "9"

      -Name "SYS_PP_TO_MAIN_PROFINET_IN" -SignalType "DI"\
      -Device "PN_Internal_Device" -DeviceMap "10"

      -Name "SYS_START_PROFINET_IN" -SignalType "DI"\
      -Device "PN_Internal_Device" -DeviceMap "11"

      -Name "SYS_STOP_PROFINET_IN" -SignalType "DI" -Device "PN_Internal_Device"\
      -DeviceMap "12"

      -Name "PLC_CMD_START_PROFINET_IN" -SignalType "DI"\
      -Device "PN_Internal_Device" -DeviceMap "16" -EncType "UNSIGNED"

      -Name "PLC_CMD_STOP_PROFINET_IN" -SignalType "DI"\
      -Device "PN_Internal_Device" -DeviceMap "17" -EncType "UNSIGNED"

      -Name "PLC_CMD_UTP_PROFINET_IN" -SignalType "DI"\
      -Device "PN_Internal_Device" -DeviceMap "18" -EncType "UNSIGNED"

      -Name "PLC_CMD_MAIN_ID_PROFINET_IN" -SignalType "GI"\
      -Device "PN_Internal_Device" -DeviceMap "24-31" -EncType "UNSIGNED"

      -Name "PLC_CMD_UPT_ID_PROFINET_IN" -SignalType "GI"\
      -Device "PN_Internal_Device" -DeviceMap "32-39" -EncType "UNSIGNED"

      -Name "PLC_TRAJ_SIZE_PROFINET_IN" -SignalType "GI"\
      -Device "PN_Internal_Device" -DeviceMap "40-55" -EncType "UNSIGNED"

      -Name "SPEED_DATA_PROFINET_IN" -SignalType "GI"\
      -Device "PN_Internal_Device" -DeviceMap "56-63" -EncType "UNSIGNED"

      -Name "ZONE_DATA_PROFINET_IN" -SignalType "GI"\
      -Device "PN_Internal_Device" -DeviceMap "64-71" -EncType "UNSIGNED"

      -Name "Q0_PROFINET_IN" -SignalType "GI" -Device "PN_Internal_Device"\
      -DeviceMap "72-87" -EncType "UNSIGNED"

      -Name "Q1_PROFINET_IN" -SignalType "GI" -Device "PN_Internal_Device"\
      -DeviceMap "88-103" -EncType "UNSIGNED"

      -Name "Q2_PROFINET_IN" -SignalType "GI" -Device "PN_Internal_Device"\
      -DeviceMap "104-119" -EncType "UNSIGNED"

      -Name "Q3_PROFINET_IN" -SignalType "GI" -Device "PN_Internal_Device"\
      -DeviceMap "120-135" -EncType "UNSIGNED"

      -Name "Q4_PROFINET_IN" -SignalType "GI" -Device "PN_Internal_Device"\
      -DeviceMap "136-151" -EncType "UNSIGNED"

      -Name "Q5_PROFINET_IN" -SignalType "GI" -Device "PN_Internal_Device"\
      -DeviceMap "152-167" -EncType "UNSIGNED"

      -Name "Q0_SIGN_PROFINET_IN" -SignalType "DI" -Device "PN_Internal_Device"\
      -DeviceMap "184" -EncType "UNSIGNED"

      -Name "Q1_SIGN_PROFINET_IN" -SignalType "DI" -Device "PN_Internal_Device"\
      -DeviceMap "185" -EncType "UNSIGNED"

      -Name "Q2_SIGN_PROFINET_IN" -SignalType "DI" -Device "PN_Internal_Device"\
      -DeviceMap "186" -EncType "UNSIGNED"

      -Name "Q3_SIGN_PROFINET_IN" -SignalType "DI" -Device "PN_Internal_Device"\
      -DeviceMap "187" -EncType "UNSIGNED"

      -Name "Q4_SIGN_PROFINET_IN" -SignalType "DI" -Device "PN_Internal_Device"\
      -DeviceMap "188" -EncType "UNSIGNED"

      -Name "Q5_SIGN_PROFINET_IN" -SignalType "DI" -Device "PN_Internal_Device"\
      -DeviceMap "189" -EncType "UNSIGNED"

      -Name "RTOOL_RH_PROFINET_IN" -SignalType "DI" -Device "PN_Internal_Device"\
      -DeviceMap "400" -EncType "UNSIGNED"

      -Name "RTOOL_X_POS_PROFINET_IN" -SignalType "GI"\
      -Device "PN_Internal_Device" -DeviceMap "408-439" -EncType "UNSIGNED"

      -Name "RTOOL_Y_POS_PROFINET_IN" -SignalType "GI"\
      -Device "PN_Internal_Device" -DeviceMap "440-471" -EncType "UNSIGNED"

      -Name "RTOOL_Z_POS_PROFINET_IN" -SignalType "GI"\
      -Device "PN_Internal_Device" -DeviceMap "472-503" -EncType "UNSIGNED"

      -Name "RTOOL_X_POS_SING_PROFINET_IN" -SignalType "DI"\
      -Device "PN_Internal_Device" -DeviceMap "504" -EncType "UNSIGNED"

      -Name "RTOOL_Y_POS_SING_PROFINET_IN" -SignalType "DI"\
      -Device "PN_Internal_Device" -DeviceMap "505" -EncType "UNSIGNED"

      -Name "RTOOL_Z_POS_SING_PROFINET_IN" -SignalType "DI"\
      -Device "PN_Internal_Device" -DeviceMap "506" -EncType "UNSIGNED"

      -Name "RTOOL_QX_ROT_PROFINET_IN" -SignalType "GI"\
      -Device "PN_Internal_Device" -DeviceMap "512-543" -EncType "UNSIGNED"

      -Name "RTOOL_QY_ROT_PROFINET_IN" -SignalType "GI"\
      -Device "PN_Internal_Device" -DeviceMap "544-575" -EncType "UNSIGNED"

      -Name "RTOOL_QZ_ROT_PROFINET_IN" -SignalType "GI"\
      -Device "PN_Internal_Device" -DeviceMap "576-607" -EncType "UNSIGNED"

      -Name "RTOOL_QW_ROT_PROFINET_IN" -SignalType "GI"\
      -Device "PN_Internal_Device" -DeviceMap "608-639" -EncType "UNSIGNED"

      -Name "RTOOL_QX_ROT_SIGN_PROFINET_IN" -SignalType "DI"\
      -Device "PN_Internal_Device" -DeviceMap "640" -EncType "UNSIGNED"

      -Name "RTOOL_QY_ROT_SIGN_PROFINET_IN" -SignalType "DI"\
      -Device "PN_Internal_Device" -DeviceMap "641" -EncType "UNSIGNED"

      -Name "RTOOL_QZ_ROT_SIGN_PROFINET_IN" -SignalType "DI"\
      -Device "PN_Internal_Device" -DeviceMap "642" -EncType "UNSIGNED"

      -Name "RTOOL_QW_ROT_SIGN_PROFINET_IN" -SignalType "DI"\
      -Device "PN_Internal_Device" -DeviceMap "643" -EncType "UNSIGNED"

      -Name "RTOOL_MASS_PROFINET_IN" -SignalType "GI"\
      -Device "PN_Internal_Device" -DeviceMap "648-663" -EncType "UNSIGNED"

      -Name "RTOOL_X_COG_PROFINET_IN" -SignalType "GI"\
      -Device "PN_Internal_Device" -DeviceMap "664-695" -EncType "UNSIGNED"

      -Name "RTOOL_Y_COG_PROFINET_IN" -SignalType "GI"\
      -Device "PN_Internal_Device" -DeviceMap "696-727" -EncType "UNSIGNED"

      -Name "RTOOL_Z_COG_PROFINET_IN" -SignalType "GI"\
      -Device "PN_Internal_Device" -DeviceMap "728-759" -EncType "UNSIGNED"

      -Name "RTOOL_X_COG_SIGN_PROFINET_IN" -SignalType "DI"\
      -Device "PN_Internal_Device" -DeviceMap "760" -EncType "UNSIGNED"

      -Name "RTOOL_Y_COG_SIGN_PROFINET_IN" -SignalType "DI"\
      -Device "PN_Internal_Device" -DeviceMap "761" -EncType "UNSIGNED"

      -Name "RTOOL_Z_COG_SIGN_PROFINET_IN" -SignalType "DI"\
      -Device "PN_Internal_Device" -DeviceMap "762" -EncType "UNSIGNED"

      -Name "RTOOL_QX_AOM_PROFINET_IN" -SignalType "GI"\
      -Device "PN_Internal_Device" -DeviceMap "768-799" -EncType "UNSIGNED"

      -Name "RTOOL_QY_AOM_PROFINET_IN" -SignalType "GI"\
      -Device "PN_Internal_Device" -DeviceMap "800-831" -EncType "UNSIGNED"

      -Name "RTOOL_QZ_AOM_PROFINET_IN" -SignalType "GI"\
      -Device "PN_Internal_Device" -DeviceMap "832-863" -EncType "UNSIGNED"

      -Name "RTOOL_QW_AOM_PROFINET_IN" -SignalType "GI"\
      -Device "PN_Internal_Device" -DeviceMap "864-895" -EncType "UNSIGNED"

      -Name "RTOOL_QX_AOM_SIGN_PROFINET_IN" -SignalType "DI"\
      -Device "PN_Internal_Device" -DeviceMap "896" -EncType "UNSIGNED"

      -Name "RTOOL_QY_AOM_SIGN_PROFINET_IN" -SignalType "DI"\
      -Device "PN_Internal_Device" -DeviceMap "897" -EncType "UNSIGNED"

      -Name "RTOOL_QZ_AOM_SIGN_PROFINET_IN" -SignalType "DI"\
      -Device "PN_Internal_Device" -DeviceMap "898" -EncType "UNSIGNED"

      -Name "RTOOL_QW_AOM_SIGN_PROFINET_IN" -SignalType "DI"\
      -Device "PN_Internal_Device" -DeviceMap "899" -EncType "UNSIGNED"

      -Name "RTOOL_IX_MOI_PROFINET_IN" -SignalType "GI"\
      -Device "PN_Internal_Device" -DeviceMap "904-935" -EncType "UNSIGNED"

      -Name "RTOOL_IY_MOI_PROFINET_IN" -SignalType "GI"\
      -Device "PN_Internal_Device" -DeviceMap "936-967" -EncType "UNSIGNED"

      -Name "RTOOL_IZ_MOI_PROFINET_IN" -SignalType "GI"\
      -Device "PN_Internal_Device" -DeviceMap "968-999" -EncType "UNSIGNED"

      -Name "ROB_MOTION_TRAJ_ID_PROFINET_OUT" -SignalType "GO"\
      -Device "PN_Internal_Device" -DeviceMap "32-47"

      -Name "Q6_PROFINET_OUT" -SignalType "GO" -Device "PN_Internal_Device"\
      -DeviceMap "144-159" -EncType "UNSIGNED"

      -Name "Q6_SIGN_PROFINET_OUT" -SignalType "DO" -Device "PN_Internal_Device"\
      -DeviceMap "166" -EncType "UNSIGNED"

      -Name "Q6_PROFINET_IN" -SignalType "GI" -Device "PN_Internal_Device"\
      -DeviceMap "168-183" -EncType "UNSIGNED"

      -Name "Q6_SIGN_PROFINET_IN" -SignalType "DI" -Device "PN_Internal_Device"\
      -DeviceMap "190" -EncType "UNSIGNED"

      -Name "TCP_POS_X_SIGN_PROFINET_OUT" -SignalType "DO"\
      -Device "PN_Internal_Device" -DeviceMap "328" -EncType "UNSIGNED"

      -Name "TCP_POS_Y_SIGN_PROFINET_OUT" -SignalType "DO"\
      -Device "PN_Internal_Device" -DeviceMap "329" -EncType "UNSIGNED"

      -Name "TCP_POS_Z_SIGN_PROFINET_OUT" -SignalType "DO"\
      -Device "PN_Internal_Device" -DeviceMap "330" -EncType "UNSIGNED"

      -Name "TCP_ROT_X_SIGN_PROFINET_OUT" -SignalType "DO"\
      -Device "PN_Internal_Device" -DeviceMap "331" -EncType "UNSIGNED"

      -Name "TCP_ROT_Y_SIGN_PROFINET_OUT" -SignalType "DO"\
      -Device "PN_Internal_Device" -DeviceMap "332" -EncType "UNSIGNED"

      -Name "TCP_ROT_Z_SIGN_PROFINET_OUT" -SignalType "DO"\
      -Device "PN_Internal_Device" -DeviceMap "333" -EncType "UNSIGNED"

      -Name "TCP_EX_POS_SIGN_PROFINET_OUT" -SignalType "DO"\
      -Device "PN_Internal_Device" -DeviceMap "334" -EncType "UNSIGNED"

      -Name "TCP_CFG_1_SIGN_PROFINET_OUT" -SignalType "DO"\
      -Device "PN_Internal_Device" -DeviceMap "368" -EncType "UNSIGNED"

      -Name "TCP_CFG_4_SIGN_PROFINET_OUT" -SignalType "DO"\
      -Device "PN_Internal_Device" -DeviceMap "369" -EncType "UNSIGNED"

      -Name "TCP_CFG_6_SIGN_PROFINET_OUT" -SignalType "DO"\
      -Device "PN_Internal_Device" -DeviceMap "370" -EncType "UNSIGNED"

      -Name "TCP_CFG_X_SIGN_PROFINET_OUT" -SignalType "DO"\
      -Device "PN_Internal_Device" -DeviceMap "371" -EncType "UNSIGNED"

      -Name "TCP_POS_X_PROFINET_IN" -SignalType "GI"\
      -Device "PN_Internal_Device" -DeviceMap "192-223" -EncType "UNSIGNED"

      -Name "TCP_POS_Y_PROFINET_IN" -SignalType "GI"\
      -Device "PN_Internal_Device" -DeviceMap "224-255" -EncType "UNSIGNED"

      -Name "TCP_POS_Z_PROFINET_IN" -SignalType "GI"\
      -Device "PN_Internal_Device" -DeviceMap "256-287" -EncType "UNSIGNED"

      -Name "TCP_ROT_X_PROFINET_IN" -SignalType "GI"\
      -Device "PN_Internal_Device" -DeviceMap "288-303" -EncType "UNSIGNED"

      -Name "TCP_ROT_Y_PROFINET_IN" -SignalType "GI"\
      -Device "PN_Internal_Device" -DeviceMap "304-319" -EncType "UNSIGNED"

      -Name "TCP_ROT_Z_PROFINET_IN" -SignalType "GI"\
      -Device "PN_Internal_Device" -DeviceMap "320-335" -EncType "UNSIGNED"

      -Name "TCP_EX_POS_PROFINET_IN" -SignalType "GI"\
      -Device "PN_Internal_Device" -DeviceMap "336-351" -EncType "UNSIGNED"

      -Name "TCP_POS_X_SIGN_PROFINET_IN" -SignalType "DI"\
      -Device "PN_Internal_Device" -DeviceMap "352" -EncType "UNSIGNED"

      -Name "TCP_POS_Y_SIGN_PROFINET_IN" -SignalType "DI"\
      -Device "PN_Internal_Device" -DeviceMap "353" -EncType "UNSIGNED"

      -Name "TCP_POS_Z_SIGN_PROFINET_IN" -SignalType "DI"\
      -Device "PN_Internal_Device" -DeviceMap "354" -EncType "UNSIGNED"

      -Name "TCP_ROT_X_SIGN_PROFINET_IN" -SignalType "DI"\
      -Device "PN_Internal_Device" -DeviceMap "355" -EncType "UNSIGNED"

      -Name "TCP_ROT_Y_SIGN_PROFINET_IN" -SignalType "DI"\
      -Device "PN_Internal_Device" -DeviceMap "356" -EncType "UNSIGNED"

      -Name "TCP_ROT_Z_SIGN_PROFINET_IN" -SignalType "DI"\
      -Device "PN_Internal_Device" -DeviceMap "357" -EncType "UNSIGNED"

      -Name "TCP_EX_POS_SIGN_PROFINET_IN" -SignalType "DI"\
      -Device "PN_Internal_Device" -DeviceMap "358" -EncType "UNSIGNED"

      -Name "TCP_CFG_1_PROFINET_IN" -SignalType "GI"\
      -Device "PN_Internal_Device" -DeviceMap "360-367" -EncType "UNSIGNED"

      -Name "TCP_CFG_4_PROFINET_IN" -SignalType "GI"\
      -Device "PN_Internal_Device" -DeviceMap "360-367" -EncType "UNSIGNED"

      -Name "TCP_CFG_6_PROFINET_IN" -SignalType "GI"\
      -Device "PN_Internal_Device" -DeviceMap "360-367" -EncType "UNSIGNED"

      -Name "TCP_CFG_X_PROFINET_IN" -SignalType "GI"\
      -Device "PN_Internal_Device" -DeviceMap "360-367" -EncType "UNSIGNED"

      -Name "TCP_CFG_1_SIGN_PROFINET_IN" -SignalType "DI"\
      -Device "PN_Internal_Device" -DeviceMap "368" -EncType "UNSIGNED"

      -Name "TCP_CFG_4_SIGN_PROFINET_IN" -SignalType "DI"\
      -Device "PN_Internal_Device" -DeviceMap "369" -EncType "UNSIGNED"

      -Name "TCP_CFG_6_SIGN_PROFINET_IN" -SignalType "DI"\
      -Device "PN_Internal_Device" -DeviceMap "370" -EncType "UNSIGNED"

      -Name "TCP_CFG_X_SIGN_PROFINET_IN" -SignalType "DI"\
      -Device "PN_Internal_Device" -DeviceMap "371" -EncType "UNSIGNED"

      -Name "TCP_POS_X_PROFINET_OUT" -SignalType "GO"\
      -Device "PN_Internal_Device" -DeviceMap "168-199" -EncType "UNSIGNED"

      -Name "TCP_POS_Y_PROFINET_OUT" -SignalType "GO"\
      -Device "PN_Internal_Device" -DeviceMap "200-231" -EncType "UNSIGNED"

      -Name "TCP_POS_Z_PROFINET_OUT" -SignalType "GO"\
      -Device "PN_Internal_Device" -DeviceMap "232-263" -EncType "UNSIGNED"

      -Name "TCP_ROT_X_PROFINET_OUT" -SignalType "GO"\
      -Device "PN_Internal_Device" -DeviceMap "264-279" -EncType "UNSIGNED"

      -Name "TCP_ROT_Y_PROFINET_OUT" -SignalType "GO"\
      -Device "PN_Internal_Device" -DeviceMap "280-295" -EncType "UNSIGNED"

      -Name "TCP_ROT_Z_PROFINET_OUT" -SignalType "GO"\
      -Device "PN_Internal_Device" -DeviceMap "296-311" -EncType "UNSIGNED"

      -Name "TCP_EX_POS_PROFINET_OUT" -SignalType "GO"\
      -Device "PN_Internal_Device" -DeviceMap "312-327" -EncType "UNSIGNED"

      -Name "TCP_CFG_1_PROFINET_OUT" -SignalType "GO"\
      -Device "PN_Internal_Device" -DeviceMap "336-343" -EncType "UNSIGNED"

      -Name "TCP_CFG_4_PROFINET_OUT" -SignalType "GO"\
      -Device "PN_Internal_Device" -DeviceMap "344-351" -EncType "UNSIGNED"

      -Name "TCP_CFG_6_PROFINET_OUT" -SignalType "GO"\
      -Device "PN_Internal_Device" -DeviceMap "352-359" -EncType "UNSIGNED"

      -Name "TCP_CFG_X_PROFINET_OUT" -SignalType "GO"\
      -Device "PN_Internal_Device" -DeviceMap "360-367" -EncType "UNSIGNED"
